// TIA Portal V19 export
TYPE "LubrValve_Par"
// stored: Access Published
   STRUCT
      SystemOn : Bool;   // FALSE: System disabled
      EnableCheckFdbk : Bool;   // Enable Check cycle feedback
      CycleFdbkCheckTime : Time;   // Check feedback time with WorkMode=0
      WorkTime : Time;   // Work time in with WorkMode=1
      ValveONTime : Time;   // Valve ON time with VlaveType=TRUE
      ValveOFFTime : Time;   // Valve OFF time with VlaveType=TRUE
      ValvePumpSetPoint : Int;   // Quantity of ON-OFF pump with WorkMode=2
      LubrReqSetPoint : LReal;   // Space in 'm' or Operation Setpoint (see Config)
   END_STRUCT;
END_TYPE
